// Mitsubishi GX Works2 project: group_5_ex_2   PLC: FX3G

// global labels: Global1
VAR_GLOBAL
  COOKIE_REG AT D1100 : REAL;
  CREAM_REG AT D1110 : REAL;
  CHOCOLATE_REG AT D1120 : REAL;
  Start_Day AT X007 : BOOL;
  System_On AT Y007 : BOOL;
  Start_Condition AT M7 : BOOL;
END_VAR
VAR_GLOBAL CONSTANT
  CREAM_MIN_CONST : REAL := 300;
  CHOCOLATE_MIN_CONST : REAL := 240;
  COOKIE_MIN_CONST : REAL := 6.0;
END_VAR
VAR_GLOBAL
  Stop_Condition AT M1 : BOOL;
  Check_Stock AT M2 : BOOL;
  Finish_Cream_stage AT M3 : BOOL;
  Sprinkling_Stage AT X011 : BOOL;
END_VAR
VAR_GLOBAL CONSTANT
  Chocolate_Lot : REAL := 120;
  Cookie_Lot : REAL := 6.0;
  Cream_Lot : REAL := 300;
  Double_Chocolate_Lot : REAL := 240;
END_VAR
VAR_GLOBAL
  Finish_Dipping_Stage AT M5 : BOOL;
  Moving_Stage_Finish AT M4 : BOOL;
  Light_Bulb_1 AT M383 : BOOL;
  Light_Bulb_2 AT M382 : BOOL;
  Light_Bulb_Help AT M381 : BOOL;
  Flick_timer_1 AT TC0 : BOOL;
  Flick_timer_2 AT TC1 : BOOL;
END_VAR
VAR_GLOBAL CONSTANT
  Constant_Flicking_1 : INT := 6;
END_VAR
VAR_GLOBAL
  Timer_Value_1 AT TS0 : BOOL;
  Timer_Value_2 AT TS1 : BOOL;
  Timer_Value_3 AT TS2 : BOOL;
  Moving_Timer AT TC2 : BOOL;
  Moving_Flicker_light_1 AT Y001 : BOOL;
  Moving_Flicker_light_2 AT Y000 : BOOL;
  OOO AT Y011 : BOOL;
END_VAR
VAR_GLOBAL CONSTANT
  Moving_TIme : INT := 40;
END_VAR
VAR_GLOBAL
  Cream_Machine_On AT M384 : BOOL;
  Cream_Stage_On AT Y004 : BOOL;
  Dipping_Stage AT Y003 : BOOL;
  Sprinkling_On AT X010 : BOOL;
  Sen_15 AT X003 : BOOL;
  Sen_30 AT X004 : BOOL;
  Sen_Cookies_In AT X002 : BOOL;
  Sen_Cookies_FinishCam AT X001 : BOOL;
  Stop_Button AT X005 : BOOL;
  SPRINKLING_REG AT D1112 : REAL;
  DIPPING_REG AT D1122 : REAL;
  Sample_Analog_1 AT X006 : BOOL;
  Sample_Input AT D8280 : INT;
  Dipping_Type AT D1130 : INT;
END_VAR
VAR_GLOBAL CONSTANT
  More_Than_5 : INT := 5;
  Double_Dipping : INT := 10;
END_VAR
VAR_GLOBAL
  Dipping_Timer AT TC3 : BOOL;
  Dipping_Stage_On AT M380 : BOOL;
END_VAR
VAR_GLOBAL CONSTANT
  Dippinng_Time : INT := 50;
END_VAR
VAR_GLOBAL
  Dipping_Timer_Value AT TS3 : BOOL;
END_VAR
VAR_GLOBAL CONSTANT
  Converting_Analog : INT := 390;
  Less_Than_6 : INT := 6;
END_VAR
VAR_GLOBAL
  Filling_Sprinkling_reg AT M379 : BOOL;
  Test AT Y006 : BOOL;
  One_Dip_Alert AT M8 : BOOL;
  Double_Dip_Alert AT M9 : BOOL;
  Packing AT X000 : BOOL;
  Finish_Pcaking AT M6 : BOOL;
  Packing_Counter AT CC0 : BOOL;
  Packing_Counter_finish AT CS0 : BOOL;
END_VAR
VAR_GLOBAL CONSTANT
  packing_5 : INT := 5;
END_VAR
VAR_GLOBAL
  Packing_Alert AT Y002 : BOOL;
  finish_counting AT M10 : BOOL;
END_VAR
VAR_GLOBAL CONSTANT
  packing_6 : INT := 6;
END_VAR
VAR_GLOBAL
  Packing_counter_2 AT CC1 : BOOL;
  packing_counter_2_finish AT CS1 : BOOL;
  total_crembo AT D1140 : INT;
  New_Lot AT M11 : BOOL;
  Restart AT M12 : BOOL;
  End_Day_Flicker AT TC4 : BOOL;
END_VAR
VAR_GLOBAL CONSTANT
  End_Day_3 : INT := 30;
END_VAR
VAR_GLOBAL
  End_Day_Finish AT TS4 : BOOL;
  Crembo_Num AT D8282 : INT;
  Total_Crembo_To_Show AT D1150 : INT;
END_VAR
VAR_GLOBAL CONSTANT
  Constant_39 : INT := 39;
END_VAR
VAR_GLOBAL
  End_Check AT M378 : BOOL;
  input_taken AT M377 : BOOL;
  Cookie_Input AT D1160 : REAL;
  Cream_Input AT D1170 : REAL;
  Chocolate_Input AT D1180 : REAL;
END_VAR

// task Task_01 (event TRUE, interval 0, priority 31): POU_01

PROGRAM POU_01
(* structured ladder/FBD written out as ST: instructions are called as NAME(EN, inputs, outputs); _pN, _eN, _tN stand for wires *)
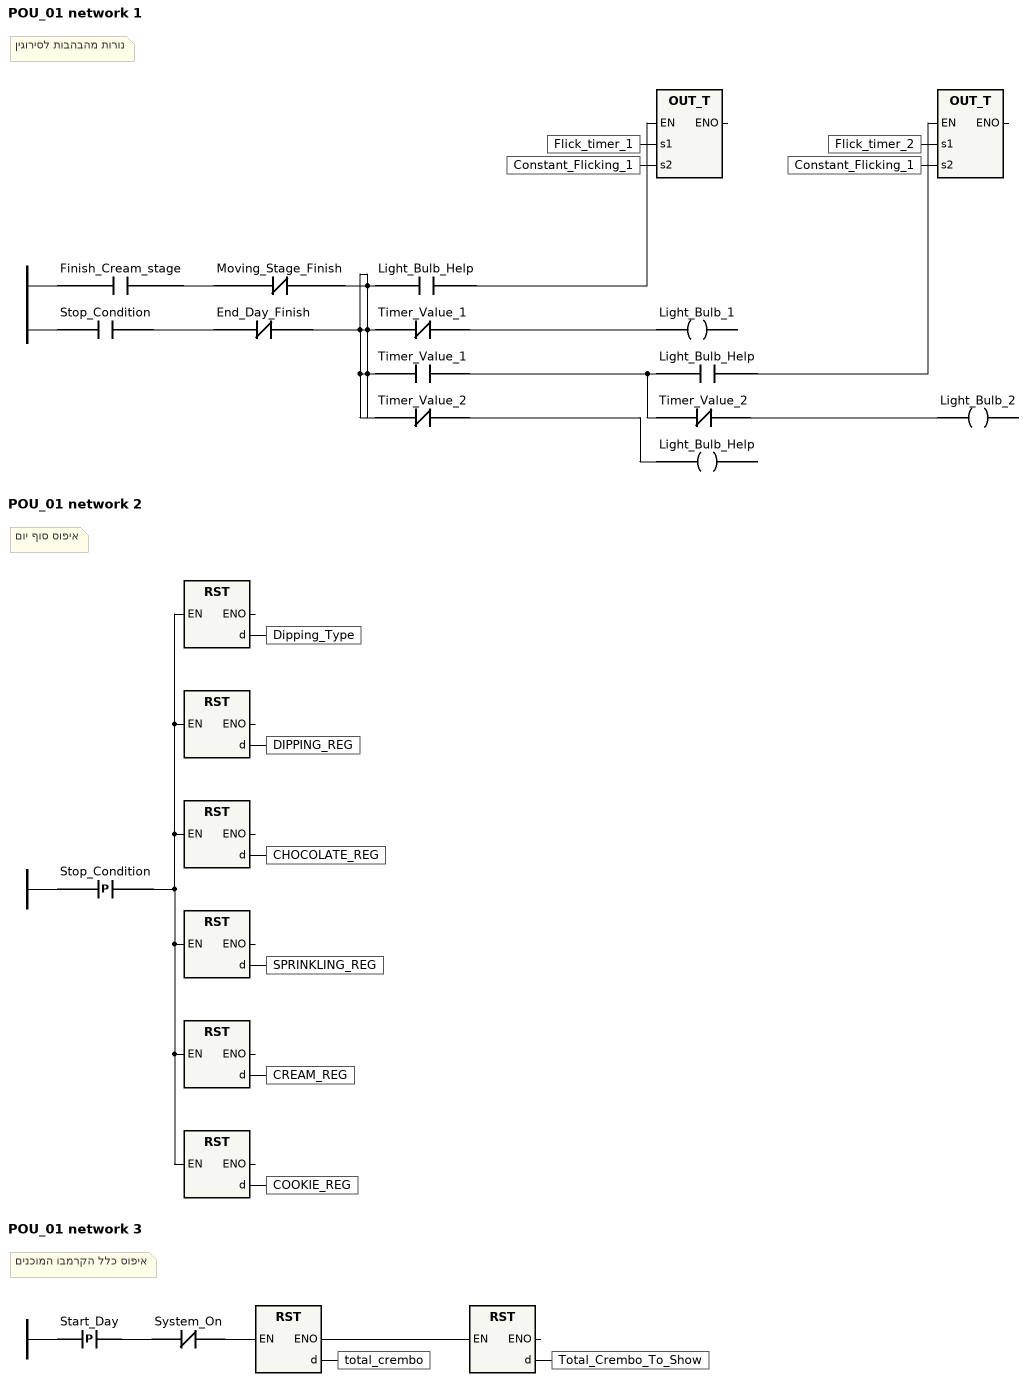
(* network 1 *)
(* נורות מהבהבות לסירוגין *)
_p1 := (Finish_Cream_stage AND NOT Moving_Stage_Finish) OR (Stop_Condition AND NOT End_Day_Finish);
OUT_T(_p1 AND Light_Bulb_Help, Flick_timer_1, Constant_Flicking_1);
Light_Bulb_1 := _p1 AND NOT Timer_Value_1;
_p2 := _p1 AND Timer_Value_1;
OUT_T(_p2 AND Light_Bulb_Help, Flick_timer_2, Constant_Flicking_1);
Light_Bulb_2 := _p2 AND NOT Timer_Value_2;
Light_Bulb_Help := _p1 AND NOT Timer_Value_2;
(* network 2 *)
(* איפוס סוף יום *)
_p1 := LDP(TRUE, Stop_Condition);
RST(_p1, Dipping_Type);
RST(_p1, DIPPING_REG);
RST(_p1, CHOCOLATE_REG);
RST(_p1, SPRINKLING_REG);
RST(_p1, CREAM_REG);
RST(_p1, COOKIE_REG);
(* network 3 *)
(* איפוס כלל הקרמבו המוכנים *)
_e1 := RST(LDP(TRUE, Start_Day) AND NOT System_On, total_crembo);
RST(_e1, Total_Crembo_To_Show);
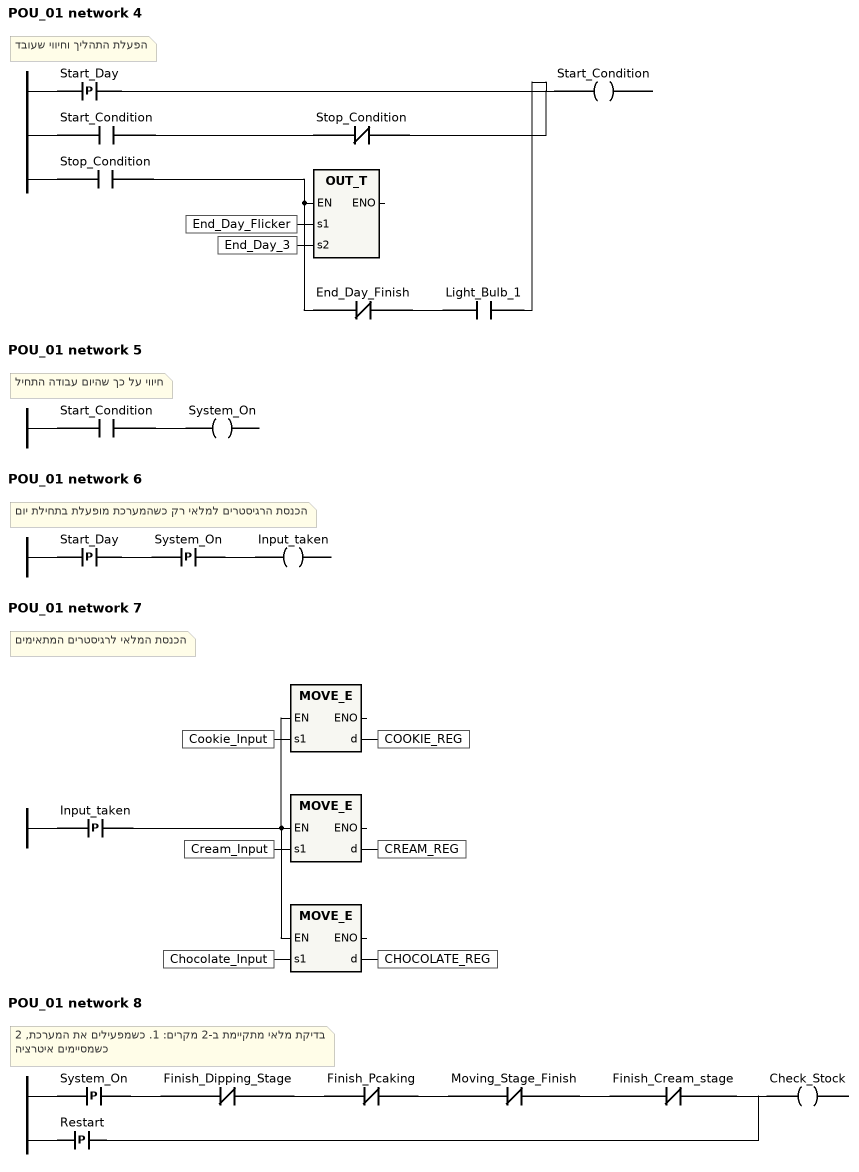
(* network 4 *)
(* הפעלת התהליך וחיווי שעובד *)
Start_Condition := LDP(TRUE, Start_Day) OR (Start_Condition AND NOT Stop_Condition) OR (Stop_Condition AND NOT End_Day_Finish AND Light_Bulb_1);
OUT_T(Stop_Condition, End_Day_Flicker, End_Day_3);
(* network 5 *)
(* חיווי על כך שהיום עבודה התחיל *)
System_On := Start_Condition;
(* network 6 *)
(* הכנסת הרגיסטרים למלאי רק כשהמערכת מופעלת בתחילת יום *)
Input_taken := LDP(TRUE, Start_Day) AND LDP(TRUE, System_On);
(* network 7 *)
(* הכנסת המלאי לרגיסטרים המתאימים *)
_p1 := LDP(TRUE, Input_taken);
MOVE_E(_p1, Cookie_Input, COOKIE_REG);
MOVE_E(_p1, Cream_Input, CREAM_REG);
MOVE_E(_p1, Chocolate_Input, CHOCOLATE_REG);
(* network 8 *)
(* בדיקת מלאי מתקיימת ב-2 מקרים: 1. כשמפעילים את המערכת, 2 כשמסיימים איטרציה *)
Check_Stock := (LDP(TRUE, System_On) AND NOT Finish_Dipping_Stage AND NOT Finish_Pcaking AND NOT Moving_Stage_Finish AND NOT Finish_Cream_stage) OR LDP(TRUE, Restart);
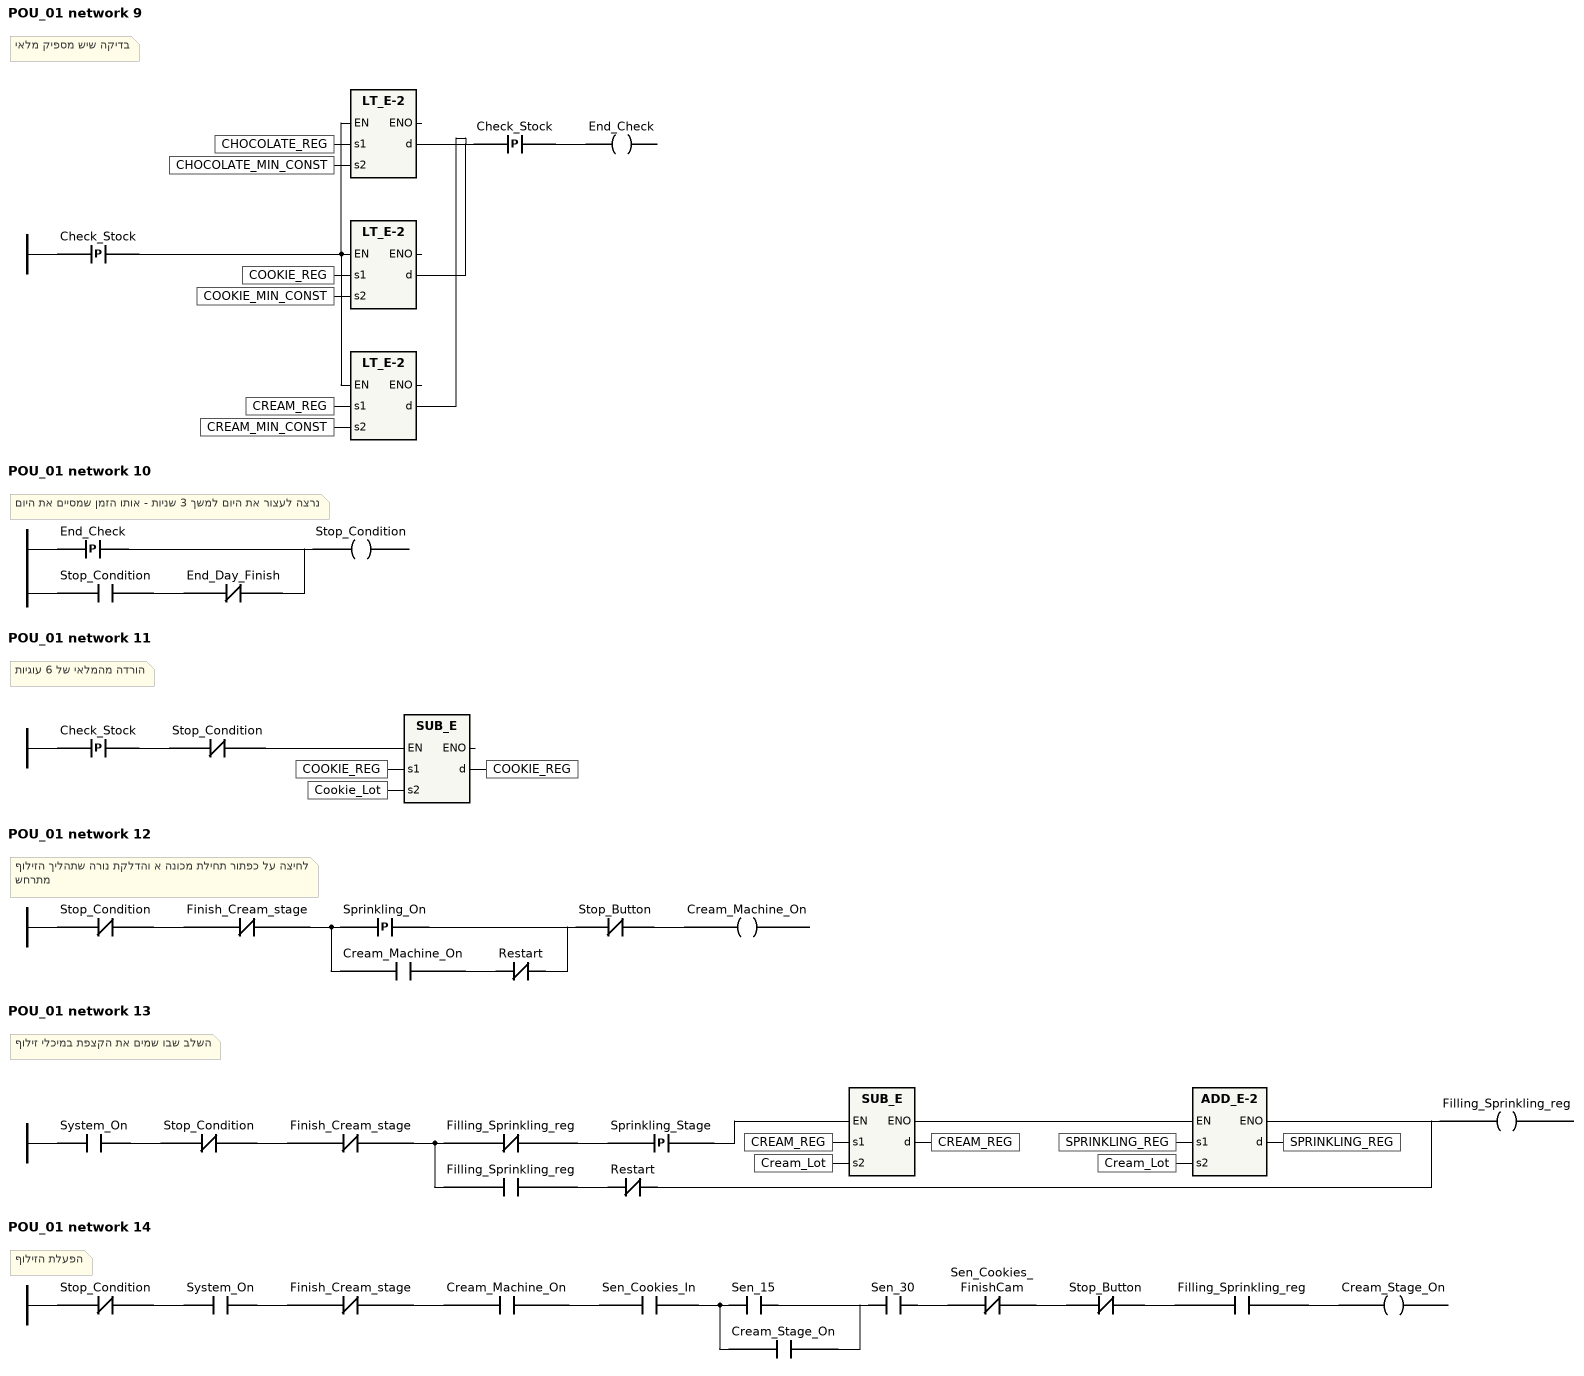
(* network 9 *)
(* בדיקה שיש מספיק מלאי *)
_p1 := LDP(TRUE, Check_Stock);
LT_E(_p1, CHOCOLATE_REG, CHOCOLATE_MIN_CONST, _t2);
LT_E(_p1, COOKIE_REG, COOKIE_MIN_CONST, _t3);
LT_E(_p1, CREAM_REG, CREAM_MIN_CONST, _t4);
End_Check := (_t2 OR _t3 OR _t4) AND LDP(TRUE, Check_Stock);
(* network 10 *)
(* נרצה לעצור את היום למשך 3 שניות - אותו הזמן שמסיים את היום *)
Stop_Condition := LDP(TRUE, End_Check) OR (Stop_Condition AND NOT End_Day_Finish);
(* network 11 *)
(* הורדה מהמלאי של 6 עוגיות *)
SUB_E(LDP(TRUE, Check_Stock) AND NOT Stop_Condition, COOKIE_REG, Cookie_Lot, COOKIE_REG);
(* network 12 *)
(* לחיצה על כפתור תחילת מכונה א והדלקת נורה שתהליך הזילוף מתרחש *)
_p1 := NOT Stop_Condition AND NOT Finish_Cream_stage;
Cream_Machine_On := ((_p1 AND LDP(TRUE, Sprinkling_On)) OR (_p1 AND Cream_Machine_On AND NOT Restart)) AND NOT Stop_Button;
(* network 13 *)
(* השלב שבו שמים את הקצפת במיכלי זילוף *)
_p1 := System_On AND NOT Stop_Condition AND NOT Finish_Cream_stage;
_e2 := SUB_E(_p1 AND NOT Filling_Sprinkling_reg AND LDP(TRUE, Sprinkling_Stage), CREAM_REG, Cream_Lot, CREAM_REG);
_e3 := ADD_E(_e2, SPRINKLING_REG, Cream_Lot, SPRINKLING_REG);
Filling_Sprinkling_reg := _e3 OR (_p1 AND Filling_Sprinkling_reg AND NOT Restart);
(* network 14 *)
(* הפעלת הזילוף *)
_p1 := NOT Stop_Condition AND System_On AND NOT Finish_Cream_stage AND Cream_Machine_On AND Sen_Cookies_In;
Cream_Stage_On := (((((_p1 AND Sen_15) OR (_p1 AND Cream_Stage_On)) AND Sen_30) AND NOT Sen_Cookies_FinishCam) AND NOT Stop_Button) AND Filling_Sprinkling_reg;
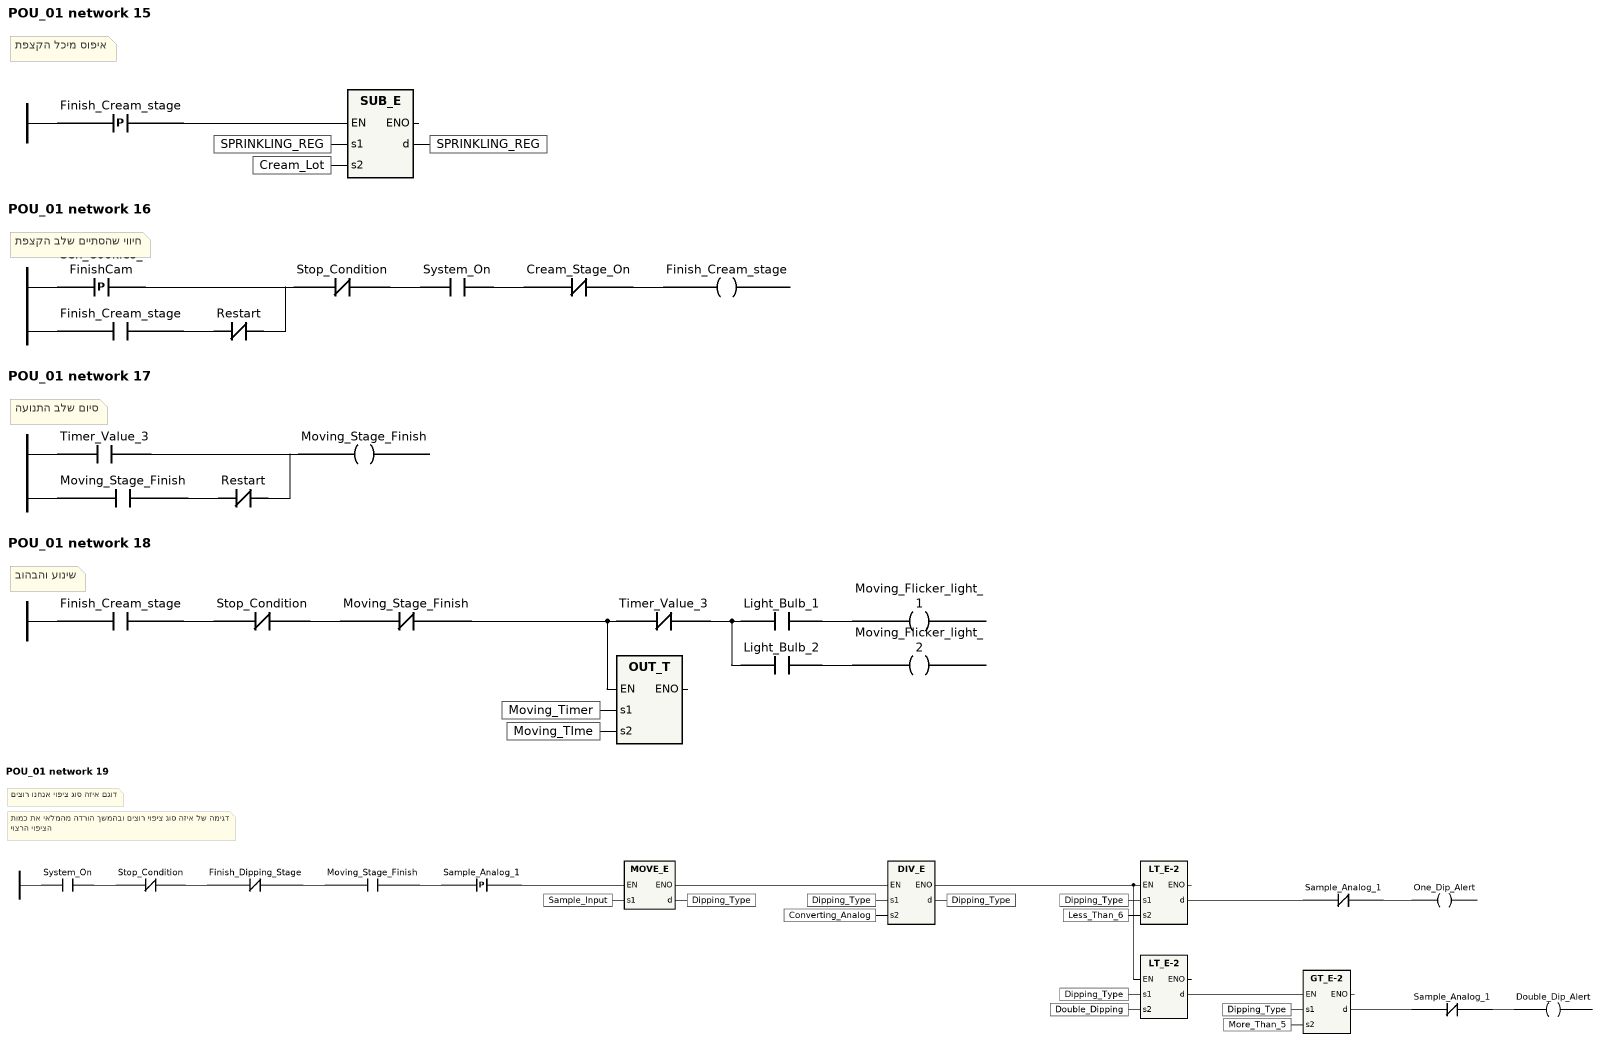
(* network 15 *)
(* איפוס מיכל הקצפת *)
SUB_E(LDP(TRUE, Finish_Cream_stage), SPRINKLING_REG, Cream_Lot, SPRINKLING_REG);
(* network 16 *)
(* חיווי שהסתיים שלב הקצפת *)
Finish_Cream_stage := (((LDP(TRUE, Sen_Cookies_FinishCam) OR (Finish_Cream_stage AND NOT Restart)) AND NOT Stop_Condition) AND System_On) AND NOT Cream_Stage_On;
(* network 17 *)
(* סיום שלב התנועה *)
Moving_Stage_Finish := Timer_Value_3 OR (Moving_Stage_Finish AND NOT Restart);
(* network 18 *)
(* שינוע והבהוב *)
_p1 := Finish_Cream_stage AND NOT Stop_Condition AND NOT Moving_Stage_Finish;
_p2 := _p1 AND NOT Timer_Value_3;
Moving_Flicker_light_1 := _p2 AND Light_Bulb_1;
OUT_T(_p1, Moving_Timer, Moving_TIme);
Moving_Flicker_light_2 := _p2 AND Light_Bulb_2;
(* network 19 *)
(* דוגם איזה סוג ציפוי אנחנו רוצים *)
(* דגימה של איזה סוג ציפוי רוצים ובהמשך הורדה מהמלאי את כמות הציפוי הרצוי *)
_e1 := MOVE_E(System_On AND NOT Stop_Condition AND NOT Finish_Dipping_Stage AND Moving_Stage_Finish AND LDP(TRUE, Sample_Analog_1), Sample_Input, Dipping_Type);
_e2 := DIV_E(_e1, Dipping_Type, Converting_Analog, Dipping_Type);
LT_E(_e2, Dipping_Type, Less_Than_6, _t3);
One_Dip_Alert := _t3 AND NOT Sample_Analog_1;
LT_E(_e2, Dipping_Type, Double_Dipping, _t4);
GT_E(_t4, Dipping_Type, More_Than_5, _t5);
Double_Dip_Alert := _t5 AND NOT Sample_Analog_1;
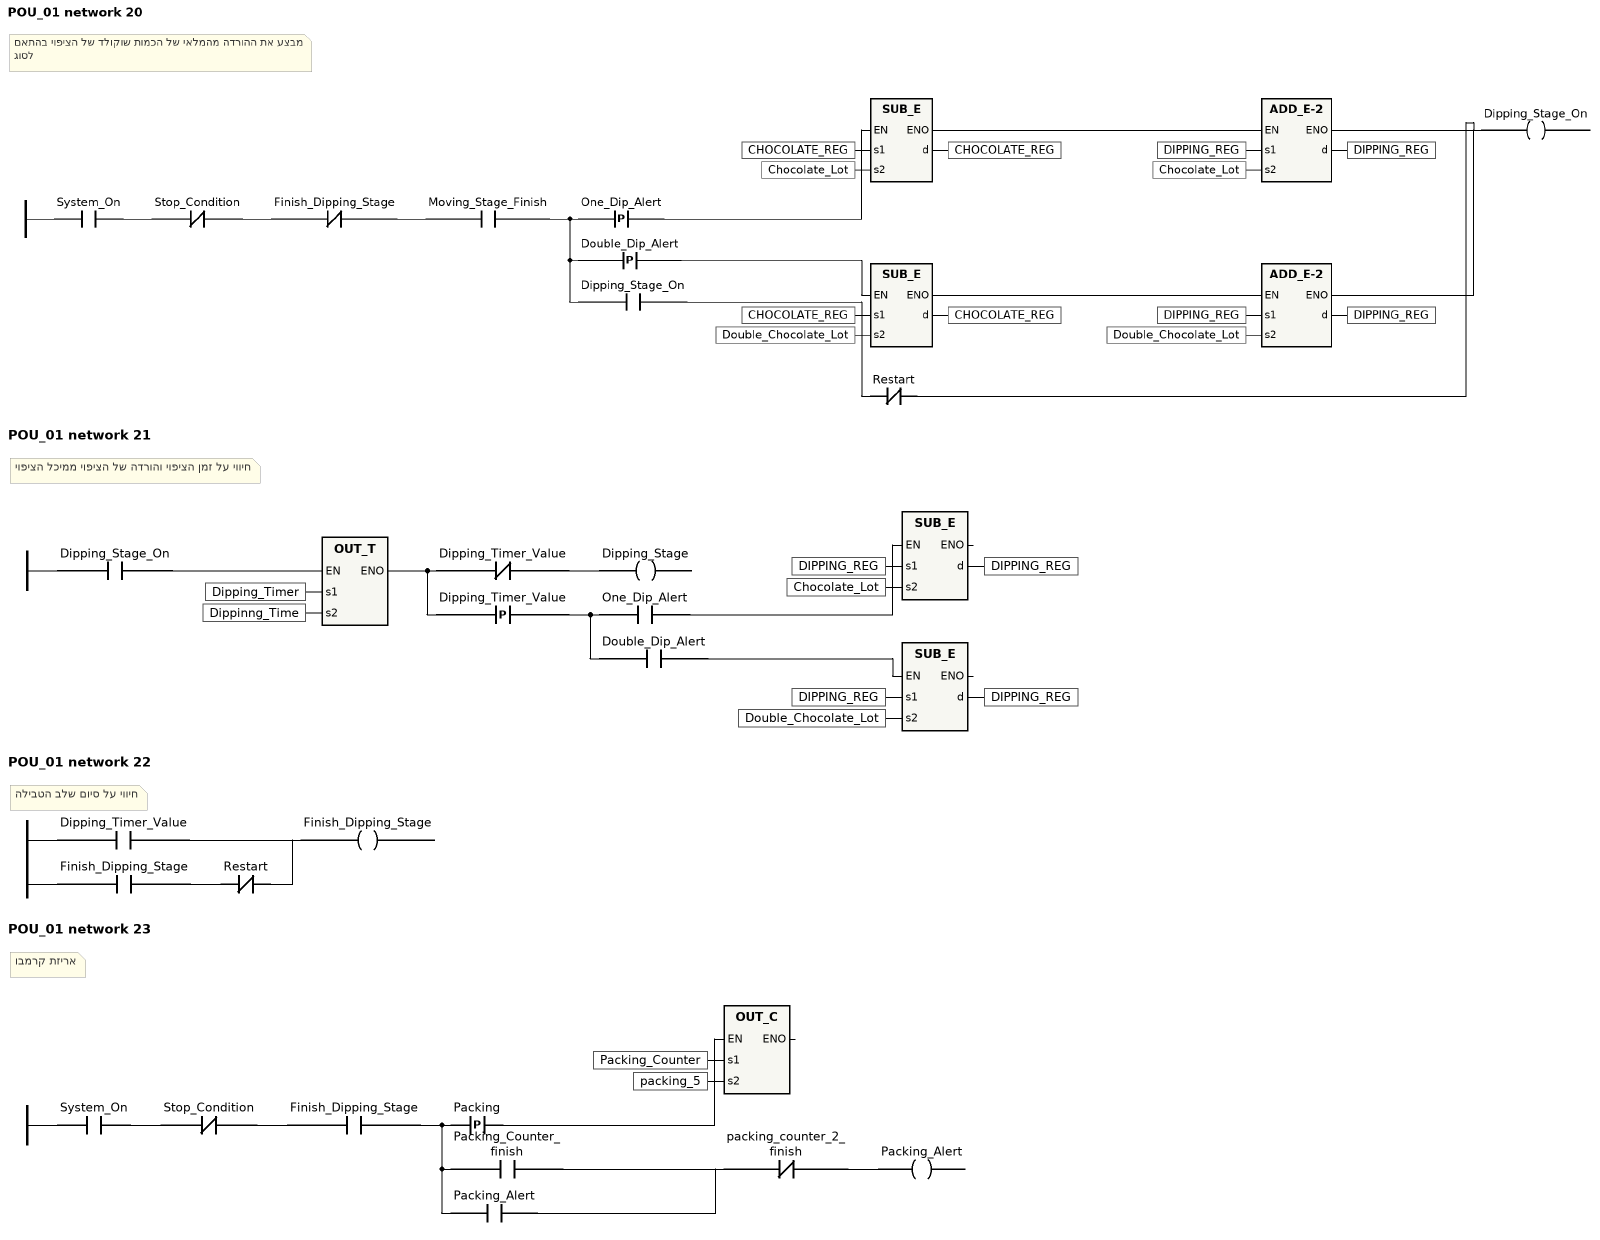
(* network 20 *)
(* מבצע את ההורדה מהמלאי של הכמות שוקולד של הציפוי בהתאם לסוג *)
_p1 := System_On AND NOT Stop_Condition AND NOT Finish_Dipping_Stage AND Moving_Stage_Finish;
_e2 := SUB_E(_p1 AND LDP(TRUE, One_Dip_Alert), CHOCOLATE_REG, Chocolate_Lot, CHOCOLATE_REG);
_e3 := ADD_E(_e2, DIPPING_REG, Chocolate_Lot, DIPPING_REG);
_e4 := SUB_E(_p1 AND LDP(TRUE, Double_Dip_Alert), CHOCOLATE_REG, Double_Chocolate_Lot, CHOCOLATE_REG);
_e5 := ADD_E(_e4, DIPPING_REG, Double_Chocolate_Lot, DIPPING_REG);
Dipping_Stage_On := _e3 OR _e5 OR (_p1 AND Dipping_Stage_On AND NOT Restart);
(* network 21 *)
(* חיווי על זמן הציפוי והורדה של הציפוי ממיכל הציפוי *)
_e1 := OUT_T(Dipping_Stage_On, Dipping_Timer, Dippinng_Time);
Dipping_Stage := _e1 AND NOT Dipping_Timer_Value;
_p2 := _e1 AND LDP(TRUE, Dipping_Timer_Value);
SUB_E(_p2 AND One_Dip_Alert, DIPPING_REG, Chocolate_Lot, DIPPING_REG);
SUB_E(_p2 AND Double_Dip_Alert, DIPPING_REG, Double_Chocolate_Lot, DIPPING_REG);
(* network 22 *)
(* חיווי על סיום שלב הטבילה *)
Finish_Dipping_Stage := Dipping_Timer_Value OR (Finish_Dipping_Stage AND NOT Restart);
(* network 23 *)
(* אריזת קרמבו *)
_p1 := System_On AND NOT Stop_Condition AND Finish_Dipping_Stage;
OUT_C(_p1 AND LDP(TRUE, Packing), Packing_Counter, packing_5);
Packing_Alert := ((_p1 AND Packing_Counter_finish) OR (_p1 AND Packing_Alert)) AND NOT packing_counter_2_finish;
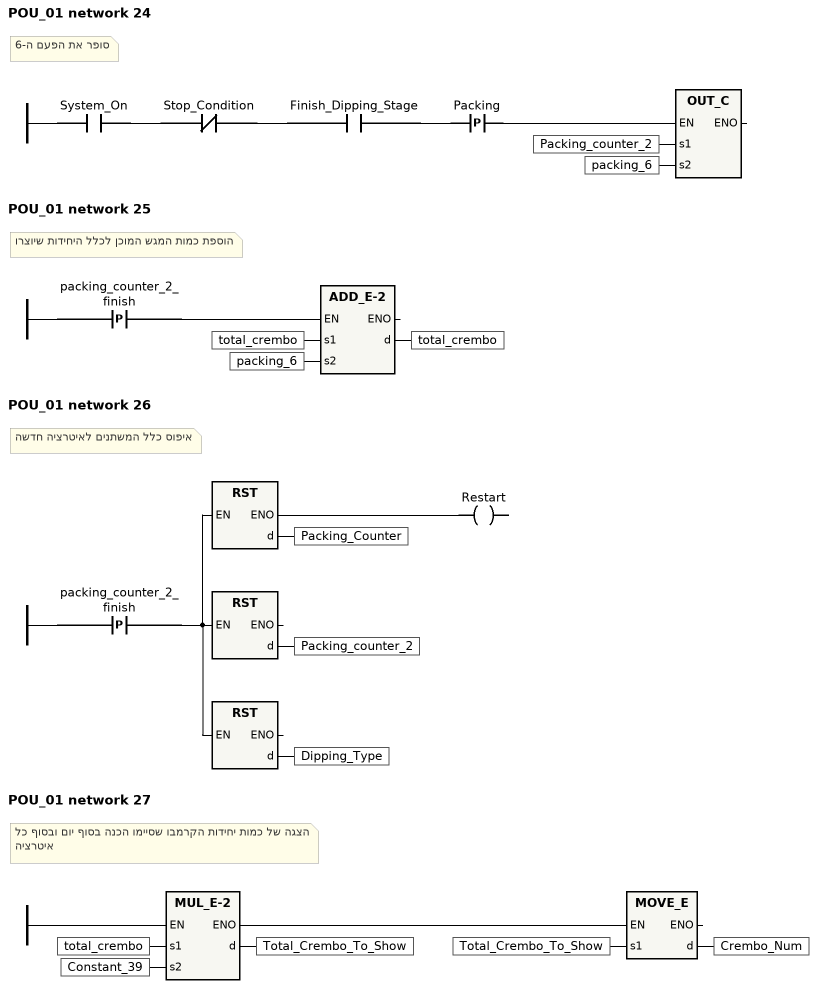
(* network 24 *)
(* סופר את הפעם ה-6 *)
OUT_C(System_On AND NOT Stop_Condition AND Finish_Dipping_Stage AND LDP(TRUE, Packing), Packing_counter_2, packing_6);
(* network 25 *)
(* הוספת כמות המגש המוכן לכלל היחידות שיוצרו *)
ADD_E(LDP(TRUE, packing_counter_2_finish), total_crembo, packing_6, total_crembo);
(* network 26 *)
(* איפוס כלל המשתנים לאיטרציה חדשה *)
_p1 := LDP(TRUE, packing_counter_2_finish);
_e2 := RST(_p1, Packing_Counter);
Restart := _e2;
RST(_p1, Packing_counter_2);
RST(_p1, Dipping_Type);
(* network 27 *)
(* הצגה של כמות יחידות הקרמבו שסיימו הכנה בסוף יום ובסוף כל איטרציה *)
_e1 := MUL_E(TRUE, total_crembo, Constant_39, Total_Crembo_To_Show);
MOVE_E(_e1, Total_Crembo_To_Show, Crembo_Num);
END_PROGRAM
